DATA_BLOCK "DB"
{ S7_Optimized_Access := 'false' }
    VAR
        p_b: BOOL;
        p_x: DINT;
        p_y: REAL;
        p_ve: BOOL;
        p_v1: DINT;
        p_v2: g_trr;
        p_v3: g_ttrrr;
        p_tv: TupleStruct2;
        p_j: DINT;
        p_r: REAL;
        p: BYTE;
        g_inp: DINT;
        p_t: REAL;
        preset_p_t: TIME;
        firstRun: BOOL;
    END_VAR
BEGIN
    firstRun := TRUE;
END_DATA_BLOCK
